REGION Network 6
   RUNG wire#powerrail
      Contact( "M_SW_AUTO" )
      "4.FC_CABINET_STATUS"()
   END_RUNG
   // the same network as SCL:
   IF "M_SW_AUTO" THEN "4.FC_CABINET_STATUS"(); END_IF;
END_REGION

REGION Network 7: FINAL FLOOR CALL CONTROL - ĐIỀU KHIỂN TẦNG GỌI CUỐI CÙNG
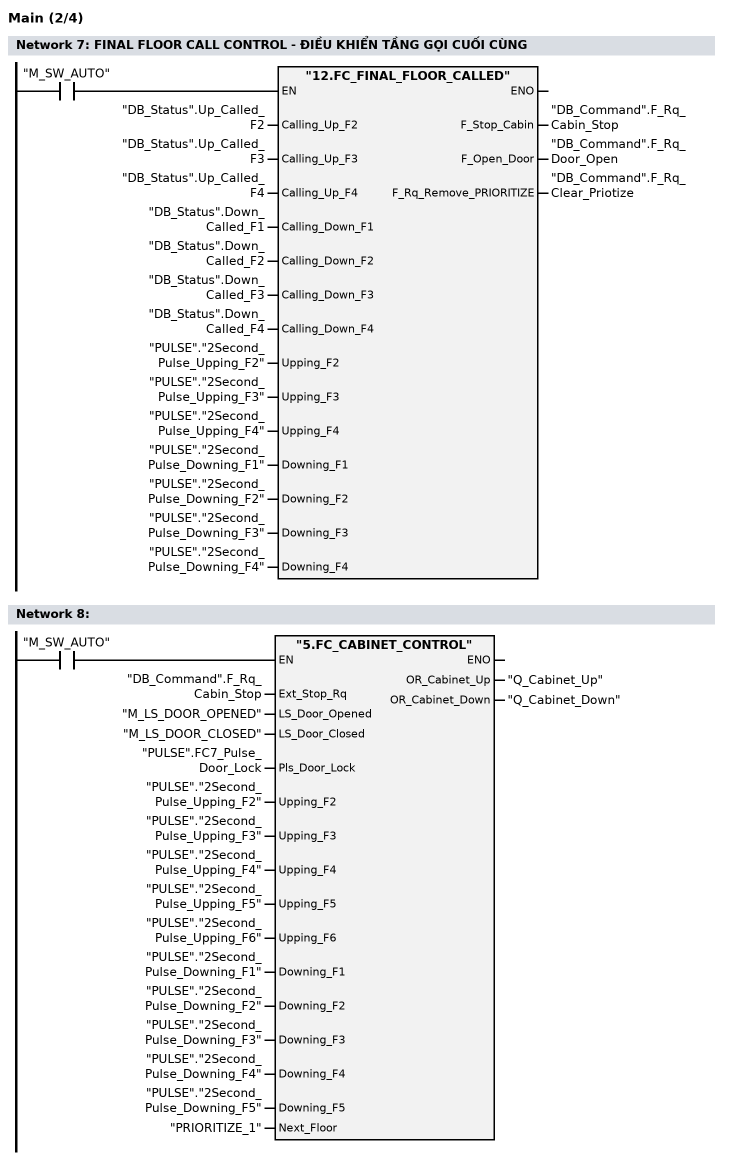
   RUNG wire#powerrail
      Contact( "M_SW_AUTO" )
      "12.FC_FINAL_FLOOR_CALLED"(Calling_Up_F2 := "DB_Status".Up_Called_F2, Calling_Up_F3 := "DB_Status".Up_Called_F3, Calling_Up_F4 := "DB_Status".Up_Called_F4, Calling_Down_F1 := "DB_Status".Down_Called_F1, Calling_Down_F2 := "DB_Status".Down_Called_F2, Calling_Down_F3 := "DB_Status".Down_Called_F3, Calling_Down_F4 := "DB_Status".Down_Called_F4, Upping_F2 := "PULSE"."2Second_Pulse_Upping_F2", Upping_F3 := "PULSE"."2Second_Pulse_Upping_F3", Upping_F4 := "PULSE"."2Second_Pulse_Upping_F4", Downing_F1 := "PULSE"."2Second_Pulse_Downing_F1", Downing_F2 := "PULSE"."2Second_Pulse_Downing_F2", Downing_F3 := "PULSE"."2Second_Pulse_Downing_F3", Downing_F4 := "PULSE"."2Second_Pulse_Downing_F4", F_Stop_Cabin => "DB_Command".F_Rq_Cabin_Stop, F_Open_Door => "DB_Command".F_Rq_Door_Open, F_Rq_Remove_PRIORITIZE => "DB_Command".F_Rq_Clear_Priotize)
   END_RUNG
   // the same network as SCL:
   IF "M_SW_AUTO" THEN
       "12.FC_FINAL_FLOOR_CALLED"(Calling_Up_F2 := "DB_Status".Up_Called_F2,
                               Calling_Up_F3 := "DB_Status".Up_Called_F3,
                               Calling_Up_F4 := "DB_Status".Up_Called_F4,
                               Calling_Down_F1 := "DB_Status".Down_Called_F1,
                               Calling_Down_F2 := "DB_Status".Down_Called_F2,
                               Calling_Down_F3 := "DB_Status".Down_Called_F3,
                               Calling_Down_F4 := "DB_Status".Down_Called_F4,
                               Upping_F2 := "PULSE"."2Second_Pulse_Upping_F2",
                               Upping_F3 := "PULSE"."2Second_Pulse_Upping_F3",
                               Upping_F4 := "PULSE"."2Second_Pulse_Upping_F4",
                               Downing_F1 := "PULSE"."2Second_Pulse_Downing_F1",
                               Downing_F2 := "PULSE"."2Second_Pulse_Downing_F2",
                               Downing_F3 := "PULSE"."2Second_Pulse_Downing_F3",
                               Downing_F4 := "PULSE"."2Second_Pulse_Downing_F4",
                               F_Stop_Cabin => "DB_Command".F_Rq_Cabin_Stop,
                               F_Open_Door => "DB_Command".F_Rq_Door_Open,
                               F_Rq_Remove_PRIORITIZE => "DB_Command".F_Rq_Clear_Priotize);
   END_IF;
END_REGION

REGION Network 8
   RUNG wire#powerrail
      Contact( "M_SW_AUTO" )
      "5.FC_CABINET_CONTROL"(Ext_Stop_Rq := "DB_Command".F_Rq_Cabin_Stop, LS_Door_Opened := "M_LS_DOOR_OPENED", LS_Door_Closed := "M_LS_DOOR_CLOSED", Pls_Door_Lock := "PULSE".FC7_Pulse_Door_Lock, Upping_F2 := "PULSE"."2Second_Pulse_Upping_F2", Upping_F3 := "PULSE"."2Second_Pulse_Upping_F3", Upping_F4 := "PULSE"."2Second_Pulse_Upping_F4", Upping_F5 := "PULSE"."2Second_Pulse_Upping_F5", Upping_F6 := "PULSE"."2Second_Pulse_Upping_F6", Downing_F1 := "PULSE"."2Second_Pulse_Downing_F1", Downing_F2 := "PULSE"."2Second_Pulse_Downing_F2", Downing_F3 := "PULSE"."2Second_Pulse_Downing_F3", Downing_F4 := "PULSE"."2Second_Pulse_Downing_F4", Downing_F5 := "PULSE"."2Second_Pulse_Downing_F5", Next_Floor := "PRIORITIZE_1", OR_Cabinet_Up => "Q_Cabinet_Up", OR_Cabinet_Down => "Q_Cabinet_Down")
   END_RUNG
   // the same network as SCL:
   IF "M_SW_AUTO" THEN
       "5.FC_CABINET_CONTROL"(Ext_Stop_Rq := "DB_Command".F_Rq_Cabin_Stop,
                              LS_Door_Opened := "M_LS_DOOR_OPENED",
                              LS_Door_Closed := "M_LS_DOOR_CLOSED",
                              Pls_Door_Lock := "PULSE".FC7_Pulse_Door_Lock,
                              Upping_F2 := "PULSE"."2Second_Pulse_Upping_F2",
                              Upping_F3 := "PULSE"."2Second_Pulse_Upping_F3",
                              Upping_F4 := "PULSE"."2Second_Pulse_Upping_F4",
                              Upping_F5 := "PULSE"."2Second_Pulse_Upping_F5",
                              Upping_F6 := "PULSE"."2Second_Pulse_Upping_F6",
                              Downing_F1 := "PULSE"."2Second_Pulse_Downing_F1",
                              Downing_F2 := "PULSE"."2Second_Pulse_Downing_F2",
                              Downing_F3 := "PULSE"."2Second_Pulse_Downing_F3",
                              Downing_F4 := "PULSE"."2Second_Pulse_Downing_F4",
                              Downing_F5 := "PULSE"."2Second_Pulse_Downing_F5",
                              Next_Floor := "PRIORITIZE_1",
                              OR_Cabinet_Up => "Q_Cabinet_Up",
                              OR_Cabinet_Down => "Q_Cabinet_Down");
   END_IF;
END_REGION

REGION Network 9: GỌI TẦNG
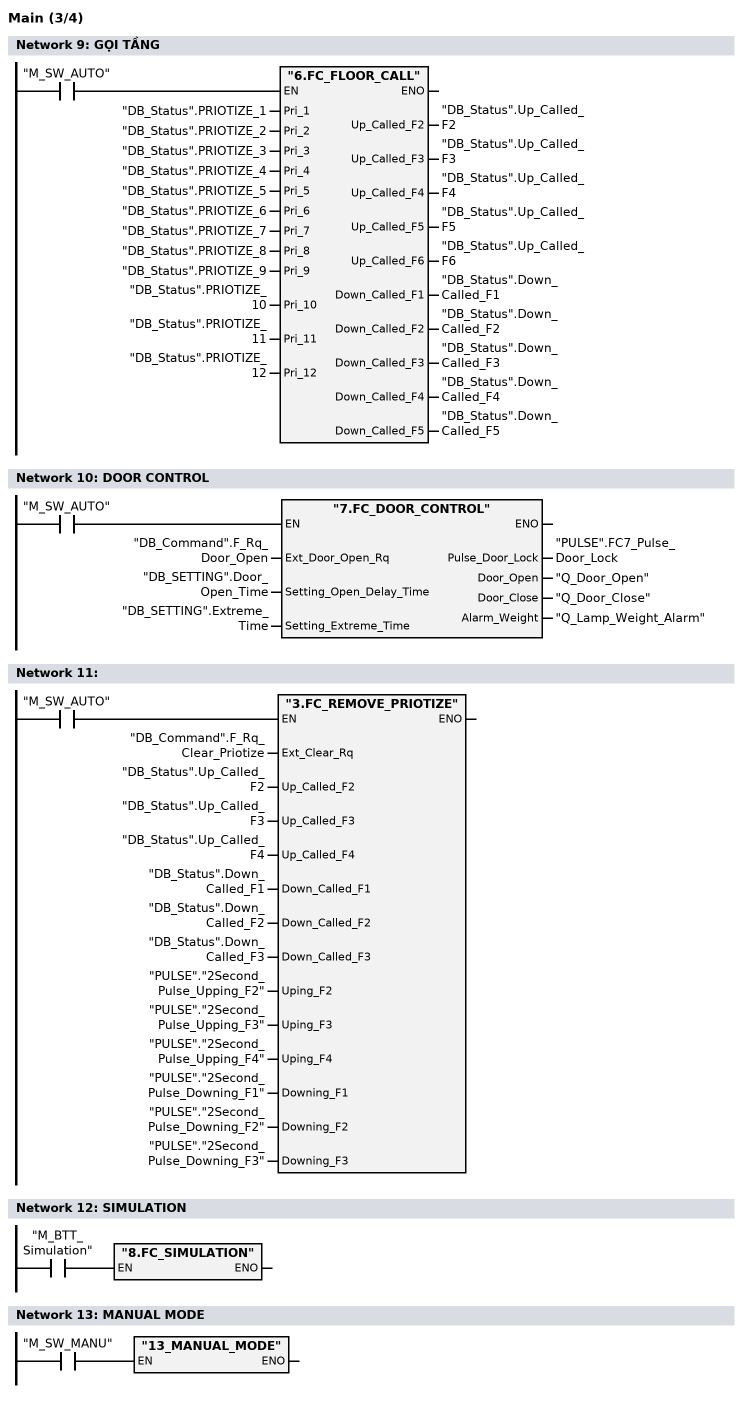
   RUNG wire#powerrail
      Contact( "M_SW_AUTO" )
      "6.FC_FLOOR_CALL"(Pri_1 := "DB_Status".PRIOTIZE_1, Pri_2 := "DB_Status".PRIOTIZE_2, Pri_3 := "DB_Status".PRIOTIZE_3, Pri_4 := "DB_Status".PRIOTIZE_4, Pri_5 := "DB_Status".PRIOTIZE_5, Pri_6 := "DB_Status".PRIOTIZE_6, Pri_7 := "DB_Status".PRIOTIZE_7, Pri_8 := "DB_Status".PRIOTIZE_8, Pri_9 := "DB_Status".PRIOTIZE_9, Pri_10 := "DB_Status".PRIOTIZE_10, Pri_11 := "DB_Status".PRIOTIZE_11, Pri_12 := "DB_Status".PRIOTIZE_12, Up_Called_F2 => "DB_Status".Up_Called_F2, Up_Called_F3 => "DB_Status".Up_Called_F3, Up_Called_F4 => "DB_Status".Up_Called_F4, Up_Called_F5 => "DB_Status".Up_Called_F5, Up_Called_F6 => "DB_Status".Up_Called_F6, Down_Called_F1 => "DB_Status".Down_Called_F1, Down_Called_F2 => "DB_Status".Down_Called_F2, Down_Called_F3 => "DB_Status".Down_Called_F3, Down_Called_F4 => "DB_Status".Down_Called_F4, Down_Called_F5 => "DB_Status".Down_Called_F5)
   END_RUNG
   // the same network as SCL:
   IF "M_SW_AUTO" THEN
       "6.FC_FLOOR_CALL"(Pri_1 := "DB_Status".PRIOTIZE_1,
                         Pri_2 := "DB_Status".PRIOTIZE_2,
                         Pri_3 := "DB_Status".PRIOTIZE_3,
                         Pri_4 := "DB_Status".PRIOTIZE_4,
                         Pri_5 := "DB_Status".PRIOTIZE_5,
                         Pri_6 := "DB_Status".PRIOTIZE_6,
                         Pri_7 := "DB_Status".PRIOTIZE_7,
                         Pri_8 := "DB_Status".PRIOTIZE_8,
                         Pri_9 := "DB_Status".PRIOTIZE_9,
                         Pri_10 := "DB_Status".PRIOTIZE_10,
                         Pri_11 := "DB_Status".PRIOTIZE_11,
                         Pri_12 := "DB_Status".PRIOTIZE_12,
                         Up_Called_F2 => "DB_Status".Up_Called_F2,
                         Up_Called_F3 => "DB_Status".Up_Called_F3,
                         Up_Called_F4 => "DB_Status".Up_Called_F4,
                         Up_Called_F5 => "DB_Status".Up_Called_F5,
                         Up_Called_F6 => "DB_Status".Up_Called_F6,
                         Down_Called_F1 => "DB_Status".Down_Called_F1,
                         Down_Called_F2 => "DB_Status".Down_Called_F2,
                         Down_Called_F3 => "DB_Status".Down_Called_F3,
                         Down_Called_F4 => "DB_Status".Down_Called_F4,
                         Down_Called_F5 => "DB_Status".Down_Called_F5);
   END_IF;
END_REGION

REGION Network 10: DOOR CONTROL
   RUNG wire#powerrail
      Contact( "M_SW_AUTO" )
      "7.FC_DOOR_CONTROL"(Ext_Door_Open_Rq := "DB_Command".F_Rq_Door_Open, Setting_Open_Delay_Time := "DB_SETTING".Door_Open_Time, Setting_Extreme_Time := "DB_SETTING".Extreme_Time, Pulse_Door_Lock => "PULSE".FC7_Pulse_Door_Lock, Door_Open => "Q_Door_Open", Door_Close => "Q_Door_Close", Alarm_Weight => "Q_Lamp_Weight_Alarm")
   END_RUNG
   // the same network as SCL:
   IF "M_SW_AUTO" THEN
       "7.FC_DOOR_CONTROL"(Ext_Door_Open_Rq := "DB_Command".F_Rq_Door_Open,
                           Setting_Open_Delay_Time := "DB_SETTING".Door_Open_Time,
                           Setting_Extreme_Time := "DB_SETTING".Extreme_Time,
                           Pulse_Door_Lock => "PULSE".FC7_Pulse_Door_Lock,
                           Door_Open => "Q_Door_Open",
                           Door_Close => "Q_Door_Close",
                           Alarm_Weight => "Q_Lamp_Weight_Alarm");
   END_IF;
END_REGION

REGION Network 11
   RUNG wire#powerrail
      Contact( "M_SW_AUTO" )
      "3.FC_REMOVE_PRIOTIZE"(Ext_Clear_Rq := "DB_Command".F_Rq_Clear_Priotize, Up_Called_F2 := "DB_Status".Up_Called_F2, Up_Called_F3 := "DB_Status".Up_Called_F3, Up_Called_F4 := "DB_Status".Up_Called_F4, Down_Called_F1 := "DB_Status".Down_Called_F1, Down_Called_F2 := "DB_Status".Down_Called_F2, Down_Called_F3 := "DB_Status".Down_Called_F3, Uping_F2 := "PULSE"."2Second_Pulse_Upping_F2", Uping_F3 := "PULSE"."2Second_Pulse_Upping_F3", Uping_F4 := "PULSE"."2Second_Pulse_Upping_F4", Downing_F1 := "PULSE"."2Second_Pulse_Downing_F1", Downing_F2 := "PULSE"."2Second_Pulse_Downing_F2", Downing_F3 := "PULSE"."2Second_Pulse_Downing_F3")
   END_RUNG
   // the same network as SCL:
   IF "M_SW_AUTO" THEN
       "3.FC_REMOVE_PRIOTIZE"(Ext_Clear_Rq := "DB_Command".F_Rq_Clear_Priotize,
                              Up_Called_F2 := "DB_Status".Up_Called_F2,
                              Up_Called_F3 := "DB_Status".Up_Called_F3,
                              Up_Called_F4 := "DB_Status".Up_Called_F4,
                              Down_Called_F1 := "DB_Status".Down_Called_F1,
                              Down_Called_F2 := "DB_Status".Down_Called_F2,
                              Down_Called_F3 := "DB_Status".Down_Called_F3,
                              Uping_F2 := "PULSE"."2Second_Pulse_Upping_F2",
                              Uping_F3 := "PULSE"."2Second_Pulse_Upping_F3",
                              Uping_F4 := "PULSE"."2Second_Pulse_Upping_F4",
                              Downing_F1 := "PULSE"."2Second_Pulse_Downing_F1",
                              Downing_F2 := "PULSE"."2Second_Pulse_Downing_F2",
                              Downing_F3 := "PULSE"."2Second_Pulse_Downing_F3");
   END_IF;
END_REGION

REGION Network 12: SIMULATION
   RUNG wire#powerrail
      Contact( "M_BTT_Simulation" )
      "8.FC_SIMULATION"()
   END_RUNG
   // the same network as SCL:
   IF "M_BTT_Simulation" THEN "8.FC_SIMULATION"(); END_IF;
END_REGION

REGION Network 13: MANUAL MODE
   RUNG wire#powerrail
      Contact( "M_SW_MANU" )
      "13_MANUAL_MODE"()
   END_RUNG
   // the same network as SCL:
   IF "M_SW_MANU" THEN "13_MANUAL_MODE"(); END_IF;
END_REGION

REGION Network 14: SET GIÁ TRỊ CÀI ĐẶT BAN ĐẦU
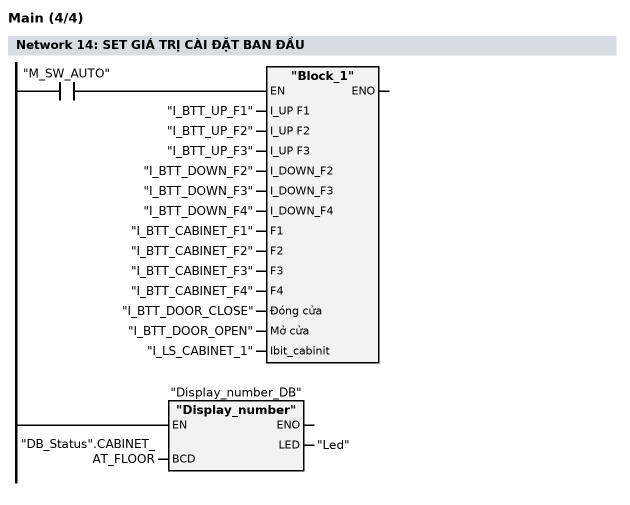
   RUNG wire#powerrail
      Contact( "M_SW_AUTO" )
      "Block_1"("I_UP F1" := "I_BTT_UP_F1", "I_UP F2" := "I_BTT_UP_F2", "I_UP F3" := "I_BTT_UP_F3", I_DOWN_F2 := "I_BTT_DOWN_F2", I_DOWN_F3 := "I_BTT_DOWN_F3", I_DOWN_F4 := "I_BTT_DOWN_F4", F1 := "I_BTT_CABINET_F1", F2 := "I_BTT_CABINET_F2", F3 := "I_BTT_CABINET_F3", F4 := "I_BTT_CABINET_F4", "Đóng cửa" := "I_BTT_DOOR_CLOSE", "Mở cửa" := "I_BTT_DOOR_OPEN", Ibit_cabinit := "I_LS_CABINET_1")
   END_RUNG
   RUNG wire#powerrail
      "Display_number_DB"(BCD := "DB_Status".CABINET_AT_FLOOR, LED => "Led")
   END_RUNG
   // the same network as SCL:
   IF "M_SW_AUTO" THEN
       "Block_1"("I_UP F1" := "I_BTT_UP_F1",
                 "I_UP F2" := "I_BTT_UP_F2",
                 "I_UP F3" := "I_BTT_UP_F3",
                 I_DOWN_F2 := "I_BTT_DOWN_F2",
                 I_DOWN_F3 := "I_BTT_DOWN_F3",
                 I_DOWN_F4 := "I_BTT_DOWN_F4",
                 F1 := "I_BTT_CABINET_F1",
                 F2 := "I_BTT_CABINET_F2",
                 F3 := "I_BTT_CABINET_F3",
                 F4 := "I_BTT_CABINET_F4",
                 "Đóng cửa" := "I_BTT_DOOR_CLOSE",
                 "Mở cửa" := "I_BTT_DOOR_OPEN",
                 Ibit_cabinit := "I_LS_CABINET_1");
   END_IF;
   "Display_number_DB"(BCD := "DB_Status".CABINET_AT_FLOOR, LED => "Led");   // "Display_number"
END_REGION
END_ORGANIZATION_BLOCK

(* ===== HMI "HMI_RT_1" =====
system functions are stored by id; their names below are inferred from use
connection "HMI_Connection_1": ETHERNET, S7_1200_OMS
connection "HMI_Connection_2": ETHERNET, S7_1200_OMS

HMI tags "Default tag table"
   "DB_SETTING_Door_Open_Time" : Time = PLC DB_SETTING.Door_Open_Time, 1 s
   "DB_SIMULATION_POS_CABINET" : Int = PLC DB_SIMULATION.POS_CABINET, 1 s
   "DB_SIMULATION_DOOR_F1" : Int = PLC DB_SIMULATION.DOOR_F1, 1 s
   "DB_SIMULATION_DOOR_F2" : Int = PLC DB_SIMULATION.DOOR_F2, 1 s
   "DB_SIMULATION_DOOR_F3" : Int = PLC DB_SIMULATION.DOOR_F3, 1 s
   "DB_SIMULATION_DOOR_F4" : Int = PLC DB_SIMULATION.DOOR_F4, 1 s
   "DB_Status_LS_F1" : Bool = PLC DB_Status.LS_F1 AT %DB1.DBX20.0, 1 s
   "DB_Status_LS_F2" : Bool = PLC DB_Status.LS_F2 AT %DB1.DBX20.1, 1 s
   "DB_Status_LS_F3" : Bool = PLC DB_Status.LS_F3 AT %DB1.DBX20.2, 1 s
   "DB_Status_LS_F4" : Bool = PLC DB_Status.LS_F4 AT %DB1.DBX20.3, 1 s
   "M_BTT_UP_F1" : Bool = PLC M_BTT_UP_F1 AT %M11.0, 1 s
   "M_BTT_UP_F2" : Bool = PLC M_BTT_UP_F2 AT %M11.1, 1 s
   "M_BTT_UP_F3" : Bool = PLC M_BTT_UP_F3 AT %M11.2, 1 s
   "M_BTT_DOWN_F2" : Bool = PLC M_BTT_DOWN_F2 AT %M11.5, 1 s
   "M_BTT_DOWN_F3" : Bool = PLC M_BTT_DOWN_F3 AT %M11.6, 1 s
   "M_BTT_DOWN_F4" : Bool = PLC M_BTT_DOWN_F4 AT %M11.7, 1 s
   "Q_BTT_Up_F1" : Bool = PLC Q_BTT_Up_F1 AT %Q0.5, 1 s
   "Q_BTT_Up_F2" : Bool = PLC Q_BTT_Up_F2 AT %Q0.6, 1 s
   "Q_BTT_Up_F3" : Bool = PLC Q_BTT_Up_F3 AT %Q0.7, 1 s
   "Q_BTT_Down_F2" : Bool = PLC Q_BTT_Down_F2 AT %Q1.2, 1 s
   "Q_BTT_Down_F3" : Bool = PLC Q_BTT_Down_F3 AT %Q1.3, 1 s
   "Q_BTT_Down_F4" : Bool = PLC Q_BTT_Down_F4 AT %Q1.4, 1 s
   "M_BTT_DOOR_OPEN" : Bool = PLC M_BTT_DOOR_OPEN AT %M10.0, 1 s
   "M_BTT_DOOR_CLOSE" : Bool = PLC M_BTT_DOOR_CLOSE AT %M10.1, 1 s
   "M_BTT_CABINET_F1" : Bool = PLC M_BTT_CABINET_F1 AT %M10.2, 1 s
   "M_BTT_CABINET_F2" : Bool = PLC M_BTT_CABINET_F2 AT %M10.3, 1 s
   "M_BTT_CABINET_F3" : Bool = PLC M_BTT_CABINET_F3 AT %M10.4, 1 s
   "M_BTT_CABINET_F4" : Bool = PLC M_BTT_CABINET_F4 AT %M10.5, 1 s
   "Q_BTT_CABIN_F1" : Bool = PLC Q_BTT_CABIN_F1 AT %Q1.7, 1 s
   "Q_BTT_CABIN_F2" : Bool = PLC Q_BTT_CABIN_F2 AT %Q2.0, 1 s
   "Q_BTT_CABIN_F3" : Bool = PLC Q_BTT_CABIN_F3 AT %Q2.1, 1 s
   "Q_BTT_CABIN_F4" : Bool = PLC Q_BTT_CABIN_F4 AT %Q2.2, 1 s
   "Q_BTT_CABIN_F5" : Bool = PLC Q_BTT_CABIN_F5 AT %Q2.3, 1 s
   "DB_SETTING_Weight" : Real = PLC DB_SETTING.Weight, 1 s
   "DB_SETTING_Extreme_Time" : Time = PLC DB_SETTING.Extreme_Time, 1 s
   "DB_SIMULATION_Weight" : DInt = PLC DB_SIMULATION.Weight, 1 s
   "Q_Lamp_System" : Bool = PLC Q_Lamp_System AT %Q0.0, 1 s
   "Q_Lamp_Weight_Alarm" : Bool = PLC Q_Lamp_Weight_Alarm AT %Q2.5, 1 s
   "M_SW_AUTO" : Bool = PLC M_SW_AUTO AT %M13.1, 1 s
   "M_SW_MANU" : Bool = PLC M_SW_MANU AT %M13.2, 1 s
   "M_BTT_Simulation" : Bool = PLC M_BTT_Simulation AT %M300.0, 1 s
   "PRIORITIZE_1" : SInt = PLC PRIORITIZE_1 AT %MB50, 1 s
   "PRIORITIZE_2" : SInt = PLC PRIORITIZE_2 AT %MB51, 1 s
   "PRIORITIZE_3" : SInt = PLC PRIORITIZE_3 AT %MB52, 1 s
   "PRIORITIZE_4" : SInt = PLC PRIORITIZE_4 AT %MB53, 1 s
   "DB_Status_CABINET_AT_FLOOR" : Int = PLC DB_Status.CABINET_AT_FLOOR AT %DB1.DBW26, 1 s
   "M_LS_DOOR_CLOSED" : Bool = PLC M_LS_DOOR_CLOSED AT %M12.4, 1 s
   "M_LS_DOOR_OPENED" : Bool = PLC M_LS_DOOR_OPENED AT %M12.3, 1 s
   "M_BTT_MAN_CABINET_UP" : Bool = PLC M_BTT_MAN_CABINET_UP AT %M12.5, 1 s
   "M_BTT_MAN_CABINET_DOWN" : Bool = PLC M_BTT_MAN_CABINET_DOWN AT %M12.6, 1 s
   "M_BTT_MAN_DOOR_OPEN" : Bool = PLC M_BTT_MAN_DOOR_OPEN AT %M12.7, 1 s
   "M_BTT_MAN_DOOR_CLOSE" : Bool = PLC M_BTT_MAN_DOOR_CLOSE AT %M13.0, 1 s
   "M_BTT_MAN_DOOR_STOP" : Bool = PLC M_BTT_MAN_DOOR_STOP AT %M13.4, 1 s
   "M_BTT_MAN_CABIN_STOP" : Bool = PLC M_BTT_MAN_CABIN_STOP AT %M13.3, 1 s
   "PLC_1_Q_Cabinet_Up" : Bool = PLC Q_Cabinet_Up AT %Q0.1, 1 s
   "PLC_1_Q_Cabinet_Down" : Bool = PLC Q_Cabinet_Down AT %Q0.2, 1 s
   "PLC_1_Led" : Byte = PLC Led AT %MB6, 1 s

graphic list "Up_Button": 0 'Up_Off'; 1 'Up_On'

graphic list "Down_Button": 0 'Down_Off'; 1 'Down_On'

screen "MAIN_SCR" 1280x800
   TextField "Text field_1" at 474,94 size 354x22; Text 'ĐIỀU KHIỂN VÀ GIÁM SÁT THANG MÁY 4 TẦNG'
   Rectangle "Rectangle_17" at 242,623 size 97x97
      HorizontalMovement <- "DB_SIMULATION_DOOR_F1"
   Rectangle "Rectangle_18" at 146,623 size 97x97
      HorizontalMovement <- "DB_SIMULATION_DOOR_F1"
   Rectangle "Rectangle_19" at 242,510 size 97x97
      HorizontalMovement <- "DB_SIMULATION_DOOR_F2"
   Rectangle "Rectangle_20" at 146,510 size 97x97
      HorizontalMovement <- "DB_SIMULATION_DOOR_F2"
   Rectangle "Rectangle_21" at 243,395 size 97x97
      HorizontalMovement <- "DB_SIMULATION_DOOR_F3"
   Rectangle "Rectangle_22" at 146,395 size 97x97
      HorizontalMovement <- "DB_SIMULATION_DOOR_F3"
   Rectangle "Rectangle_23" at 242,281 size 97x97
      HorizontalMovement <- "DB_SIMULATION_DOOR_F4"
   Rectangle "Rectangle_24" at 146,281 size 97x97
      HorizontalMovement <- "DB_SIMULATION_DOOR_F4"
   Button "Button_12" at 646,357 size 67x35; TextOff 'F2'
      on Press: SetBit("M_BTT_CABINET_F2")
      on Release: ResetBit("M_BTT_CABINET_F2")
      Appearance <- "Q_BTT_CABIN_F2"
   Button "Button_13" at 566,406 size 67x35; TextOff 'F3'
      on Press: SetBit("M_BTT_CABINET_F3")
      on Release: ResetBit("M_BTT_CABINET_F3")
      Appearance <- "Q_BTT_CABIN_F3"
   Button "Button_14" at 646,407 size 67x35; TextOff 'F4'
      on Press: SetBit("M_BTT_CABINET_F4")
      on Release: ResetBit("M_BTT_CABINET_F4")
      Appearance <- "Q_BTT_CABIN_F4"
   Button "Button_17" at 566,312 size 67x35; TextOff 'MỞ'
      on Press: SetBit("M_BTT_DOOR_OPEN")
      on Release: ResetBit("M_BTT_DOOR_OPEN")
      Appearance <- "M_BTT_DOOR_OPEN"
   Button "Button_18" at 646,310 size 67x35; TextOff 'ĐÓNG'
      on Press: SetBit("M_BTT_DOOR_CLOSE")
      on Release: ResetBit("M_BTT_DOOR_CLOSE")
      Appearance <- "M_BTT_DOOR_CLOSE"
   Switch "Switch_1" at 1033,312 size 169x71; CaptionText 'CHẾ ĐỘ VẬN HÀNH'; TextOff 'MANU'; TextOn 'AUTO'
      ProcessValue <- "M_SW_AUTO"
      on SwitchOn: SetBit("M_SW_AUTO"); ResetBit("M_SW_MANU")
      on SwitchOff: SetBit("M_SW_MANU"); ResetBit("M_SW_AUTO")
   TextField "Text field_22" at 818,321 size 74x22; Text 'ĐÈN BÁO'
   Circle "Circle_1" at 874,375 size 51x51
      Appearance <- "Q_Lamp_Weight_Alarm"
   Circle "Circle_2" at 786,375 size 51x51
      Appearance <- "Q_Lamp_System"
   TextField "Text field_23" at 776,427 size 76x22; Text 'ĐÈN RUN'
   TextField "Text field_24" at 871,426 size 58x22; Text 'ALARM'
   Switch "Switch_2" at 1032,393 size 169x71; TextOn 'ON'; CaptionText 'CHẾ ĐỘ MÔ PHỎNG'; TextOff 'OFF'
      ProcessValue <- "M_BTT_Simulation"
      on SwitchOn: SetBit("M_BTT_Simulation")
      on SwitchOff: ResetBit("M_BTT_Simulation")
   Rectangle "Rectangle_9" at 131,362 size 32x16
      Appearance <- "DB_Status_LS_F4"
   Group "Group" at 131,255 size 224x467
   Rectangle "Rectangle_8" at 131,476 size 32x16
      Appearance <- "DB_Status_LS_F3"
   Rectangle "Rectangle_11" at 131,590 size 32x16
      Appearance <- "DB_Status_LS_F2"
   Rectangle "Rectangle_12" at 131,704 size 32x16
      Appearance <- "DB_Status_LS_F1"
   Rectangle "Rectangle_13" at 131,722 size 32x16
      Appearance <- "M_LS_DOOR_OPENED"
   Rectangle "Rectangle_3" at 224,722 size 32x16
      Appearance <- "M_LS_DOOR_CLOSED"
   Rectangle "Rectangle_14" at 331,724 size 32x16
      Appearance <- "M_LS_DOOR_OPENED"
   Rectangle "Rectangle_16" at 716,575 size 55x14
      Appearance <- "PLC_1_Led"
   Rectangle "Rectangle_25" at 701,588 size 16x61
      Appearance <- "PLC_1_Led"
   Rectangle "Rectangle_26" at 770,588 size 16x61
      Appearance <- "PLC_1_Led"
   Rectangle "Rectangle_27" at 716,647 size 54x14
      Appearance <- "PLC_1_Led"
   Rectangle "Rectangle_28" at 701,660 size 16x61
      Appearance <- "PLC_1_Led"
   Rectangle "Rectangle_29" at 770,660 size 16x61
      Appearance <- "PLC_1_Led"
   Rectangle "Rectangle_30" at 717,720 size 54x14
      Appearance <- "PLC_1_Led"
   TextField "Text field_2" at 691,627 size 15x22; Text 'Text'
   TextField "Text field_3" at 689,537 size 87x29; Text 'Tầng số'
   TextField "Text field_4" at 512,568 size 39x27; Text 'Lên'
   TextField "Text field_5" at 496,705 size 66x27; Text 'Xuống'
   TextField "Text field_6" at 460,41 size 385x43; Text 'Trường đại học Duy Tân'
   Button "Button_9" at 566,358 size 67x35; TextOff 'F1'
      on Release: ResetBit("M_BTT_CABINET_F1")
      on Press: SetBit("M_BTT_CABINET_F1")
      Appearance <- "Q_BTT_CABIN_F1"
   Polygon "Polygon_1" at 585,568 size 60x47
      Appearance <- "PLC_1_Q_Cabinet_Up"
   Polygon "Polygon_2" at 585,687 size 60x47
      Appearance <- "PLC_1_Q_Cabinet_Down"
   Button "Button_1" at 361,652 size 37x40; TextOff 'Text'; PictureOff "Up_Arrow"; PictureList "Up_Button"
      on Press: SetBit("M_BTT_UP_F1")
      on Release: ResetBit("M_BTT_UP_F1")
      ProcessValue <- "Q_BTT_Up_F1"
      Appearance <- "M_BTT_UP_F1"
   Button "Button_2" at 361,564 size 37x40; TextOff 'Text'; PictureOff "Up_Arrow"; PictureList "Up_Button"
      on Press: SetBit("M_BTT_UP_F2")
      on Release: ResetBit("M_BTT_UP_F2")
      ProcessValue <- "Q_BTT_Up_F2"
   Button "Button_3" at 361,526 size 37x40; TextOff 'Text'; PictureOff "Down_Arrow"; PictureList "Down_Button"
      on Press: SetBit("M_BTT_DOWN_F2")
      on Release: ResetBit("M_BTT_DOWN_F2")
      ProcessValue <- "Q_BTT_Down_F2"
   Button "Button_4" at 361,452 size 37x40; TextOff 'Text'; PictureOff "Up_Arrow"; PictureList "Up_Button"
      on Press: SetBit("M_BTT_UP_F3")
      on Release: ResetBit("M_BTT_UP_F3")
      ProcessValue <- "Q_BTT_Up_F3"
   Button "Button_5" at 361,414 size 37x40; TextOff 'Text'; PictureOff "Down_Arrow"; PictureList "Down_Button"
      on Press: SetBit("M_BTT_DOWN_F3")
      on Release: ResetBit("M_BTT_DOWN_F3")
      ProcessValue <- "Q_BTT_Down_F3"
   Button "Button_7" at 361,302 size 37x40; TextOff 'Text'; PictureOff "Down_Arrow"; PictureList "Down_Button"
      on Press: SetBit("M_BTT_DOWN_F4")
      on Release: ResetBit("M_BTT_DOWN_F4")
      ProcessValue <- "Q_BTT_Down_F4"
*)